// Mitsubishi GX Works2 project: original_finalwithparam   PLC: FX3G

// global labels: Global1
VAR_GLOBAL
  start_day_switch AT X007 : BOOL;
  start_day_light AT Y007 : BOOL;
  cook_switch AT X001 : BOOL;
  cook_is_on_light AT Y001 : BOOL;
  lager_range AT M20 : BOOL;
  pilzner_range AT M19 : BOOL;
  enough_in_pil_stock AT M18 : BOOL;
END_VAR
VAR_GLOBAL CONSTANT
  con_shm_lag : REAL := 150.0;
  con_let_lag : REAL := 12.0;
  con_kash_lag : REAL := 60.0;
  con_shm_pil : REAL := 120.0;
  con_let_pil : REAL := 6.0;
  con_kash_pil : REAL := 53.0;
END_VAR
VAR_GLOBAL
  end_day_light AT M3 : BOOL;
  end_day_switch AT X011 : BOOL;
  shmarim AT D1150 : REAL;
  letet AT D1160 : REAL;
  kashut AT D1170 : REAL;
  analog_input1 AT D8280 : INT;
END_VAR
VAR_GLOBAL CONSTANT
  divide : INT := 400;
  const5 : INT := 5;
END_VAR
VAR_GLOBAL
  input1 AT D1110 : REAL;
  input2 AT D1120 : REAL;
  input3 AT D1130 : REAL;
  Enough_sh_lag AT M50 : BOOL;
  Enough_let_lag AT M51 : BOOL;
  Enough_ksh_lag AT M52 : BOOL;
  const_4 AT K40 : INT;
  Enough_let_pil AT M61 : BOOL;
  Enough_ksh_pil AT M62 : BOOL;
  Enough_sh_pil AT M60 : BOOL;
END_VAR
VAR_GLOBAL CONSTANT
  time_for_fer_const_3S : INT := 30;
  time_for_fer_const_4S : INT := 40;
END_VAR
VAR_GLOBAL
  fert_switch AT X005 : BOOL;
  M_Y3 AT M36 : BOOL;
  Y3_flash_counter AT TC3 : BOOL;
  Y3_light_on AT Y003 : BOOL;
  timer_ts3 AT TS3 : BOOL;
  Y4_flash_counter AT TC4 : BOOL;
  timer_ts4 AT TS4 : BOOL;
  Y4_light_on AT Y004 : BOOL;
  time_fer AT D1140 : INT;
  fert_flash_counter AT TC5 : BOOL;
  fert_flash_counter_ts AT TS5 : BOOL;
  storage_switch AT X002 : BOOL;
  counter_pack AT CC3 : BOOL;
  Y2_light_on AT Y002 : BOOL;
  CC3_term AT CS3 : BOOL;
  reg_pack_count AT D1402 : REAL;
END_VAR
VAR_GLOBAL CONSTANT
  pack_finish : REAL := 1.0;
END_VAR
VAR_GLOBAL
  const_40 AT E40.0 : REAL;
  reg_pack_count_after_multi AT D1404 : REAL;
  analog_output AT D8282 : INT;
  cook_timer AT TC9 : BOOL;
  cook_timer_ts9 AT TS9 : BOOL;
END_VAR
VAR_GLOBAL CONSTANT
  const6 : INT := 6;
END_VAR
VAR_GLOBAL
  help_gate_pil AT M39 : BOOL;
  help_gate_lag AT M38 : BOOL;
  pack_switch AT X000 : BOOL;
  enough_in_lager_stock AT M40 : BOOL;
END_VAR
VAR_GLOBAL CONSTANT
  con_zero : REAL;
END_VAR

// task Task_01 (event TRUE, interval 0, priority 31): POU_01

PROGRAM POU_01
(* structured ladder/FBD written out as ST: instructions are called as NAME(EN, inputs, outputs); _pN, _eN, _tN stand for wires *)
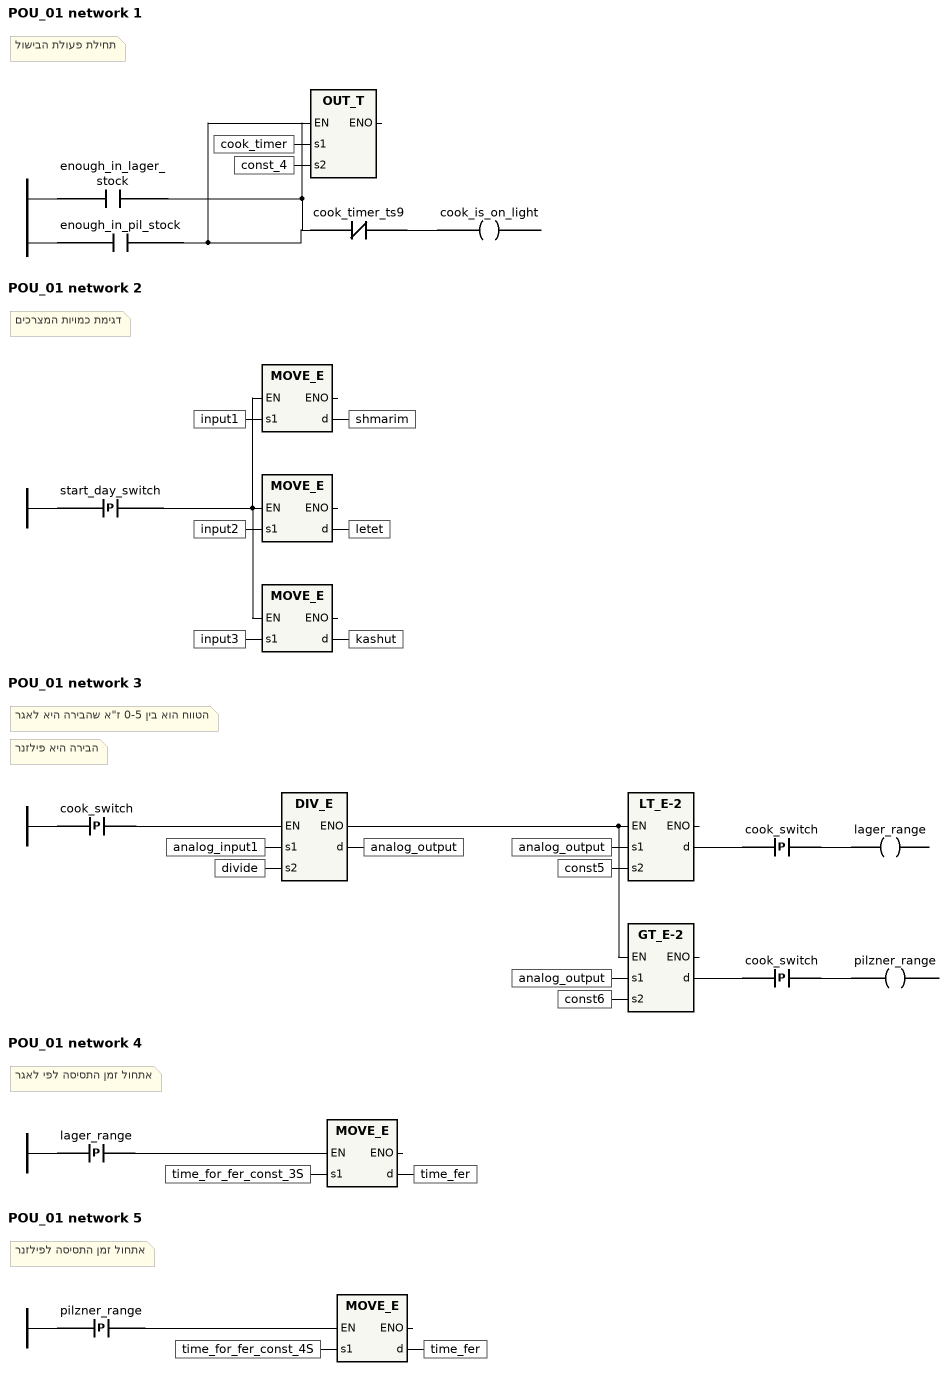
(* network 1 *)
(* תחילת פעולת הבישול *)
_p1 := enough_in_lager_stock OR enough_in_pil_stock;
OUT_T(_p1, cook_timer, const_4);
cook_is_on_light := _p1 AND NOT cook_timer_ts9;
(* network 2 *)
(* דגימת כמויות המצרכים *)
_p1 := LDP(TRUE, start_day_switch);
MOVE_E(_p1, input1, shmarim);
MOVE_E(_p1, input2, letet);
MOVE_E(_p1, input3, kashut);
(* network 3 *)
(* הטווח הוא בין 0-5 ז"א שהבירה היא לאגר *)
(* הבירה היא פילזנר *)
_e1 := DIV_E(LDP(TRUE, cook_switch), analog_input1, divide, analog_output);
LT_E(_e1, analog_output, const5, _t2);
lager_range := _t2 AND LDP(TRUE, cook_switch);
GT_E(_e1, analog_output, const6, _t3);
pilzner_range := _t3 AND LDP(TRUE, cook_switch);
(* network 4 *)
(* אתחול זמן התסיסה לפי לאגר *)
MOVE_E(LDP(TRUE, lager_range), time_for_fer_const_3S, time_fer);
(* network 5 *)
(* אתחול זמן התסיסה לפילזנר *)
MOVE_E(LDP(TRUE, pilzner_range), time_for_fer_const_4S, time_fer);
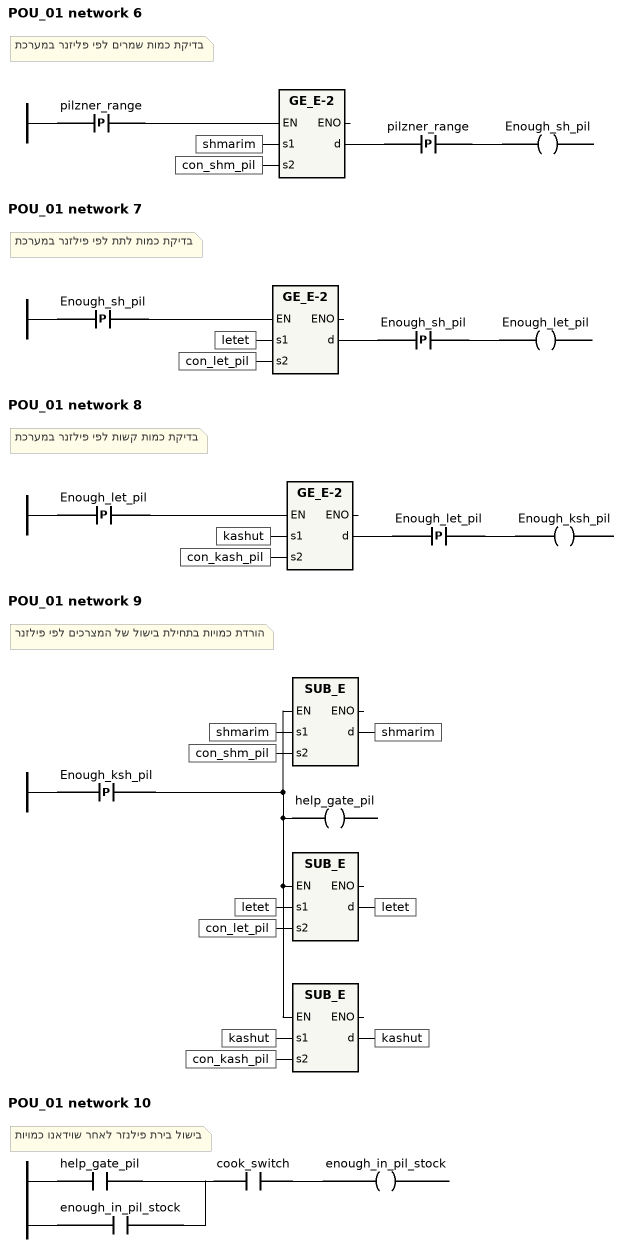
(* network 6 *)
(* בדיקת כמות שמרים לפי פליזנר במערכת *)
GE_E(LDP(TRUE, pilzner_range), shmarim, con_shm_pil, _t1);
Enough_sh_pil := _t1 AND LDP(TRUE, pilzner_range);
(* network 7 *)
(* בדיקת כמות לתת לפי פילזנר במערכת *)
GE_E(LDP(TRUE, Enough_sh_pil), letet, con_let_pil, _t1);
Enough_let_pil := _t1 AND LDP(TRUE, Enough_sh_pil);
(* network 8 *)
(* בדיקת כמות קשות לפי פילזנר במערכת *)
GE_E(LDP(TRUE, Enough_let_pil), kashut, con_kash_pil, _t1);
Enough_ksh_pil := _t1 AND LDP(TRUE, Enough_let_pil);
(* network 9 *)
(* הורדת כמויות בתחילת בישול של המצרכים לפי פילזנר *)
_p1 := LDP(TRUE, Enough_ksh_pil);
help_gate_pil := _p1;
SUB_E(_p1, shmarim, con_shm_pil, shmarim);
SUB_E(_p1, letet, con_let_pil, letet);
SUB_E(_p1, kashut, con_kash_pil, kashut);
(* network 10 *)
(* בישול בירת פילנזר לאחר שוידאנו כמויות *)
enough_in_pil_stock := (help_gate_pil OR enough_in_pil_stock) AND cook_switch;
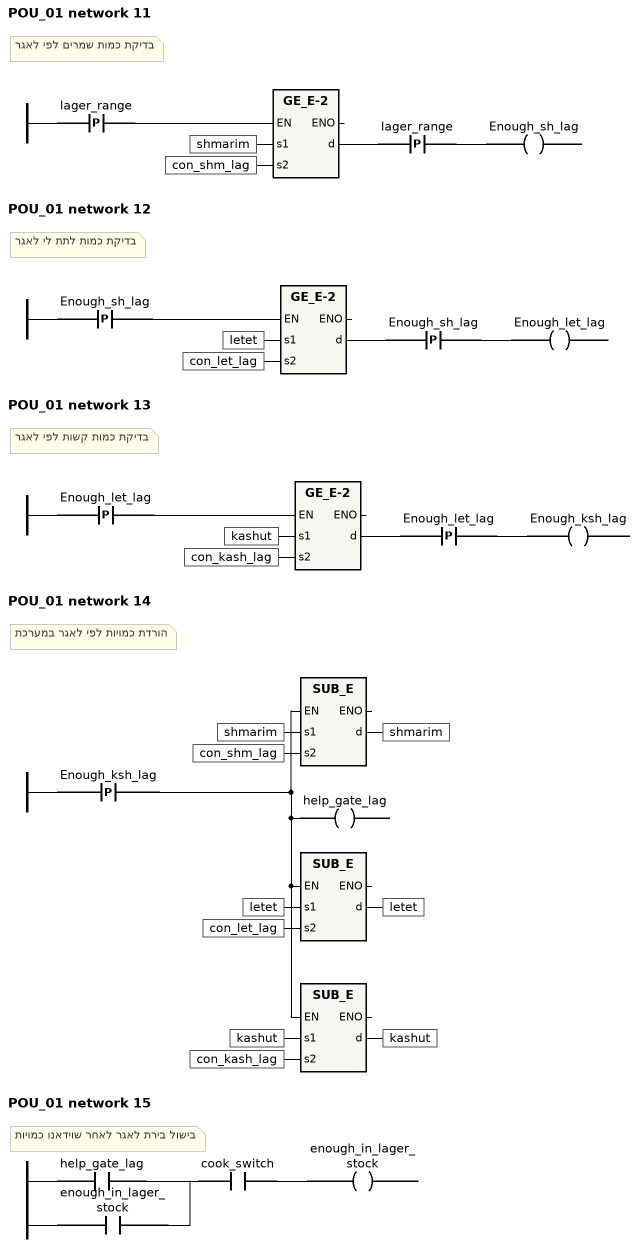
(* network 11 *)
(* בדיקת כמות שמרים לפי לאגר *)
GE_E(LDP(TRUE, lager_range), shmarim, con_shm_lag, _t1);
Enough_sh_lag := _t1 AND LDP(TRUE, lager_range);
(* network 12 *)
(* בדיקת כמות לתת לי לאגר *)
GE_E(LDP(TRUE, Enough_sh_lag), letet, con_let_lag, _t1);
Enough_let_lag := _t1 AND LDP(TRUE, Enough_sh_lag);
(* network 13 *)
(* בדיקת כמות קשות לפי לאגר *)
GE_E(LDP(TRUE, Enough_let_lag), kashut, con_kash_lag, _t1);
Enough_ksh_lag := _t1 AND LDP(TRUE, Enough_let_lag);
(* network 14 *)
(* הורדת כמויות לפי לאגר במערכת *)
_p1 := LDP(TRUE, Enough_ksh_lag);
help_gate_lag := _p1;
SUB_E(_p1, shmarim, con_shm_lag, shmarim);
SUB_E(_p1, letet, con_let_lag, letet);
SUB_E(_p1, kashut, con_kash_lag, kashut);
(* network 15 *)
(* בישול בירת לאגר לאחר שוידאנו כמויות *)
enough_in_lager_stock := (help_gate_lag OR enough_in_lager_stock) AND cook_switch;
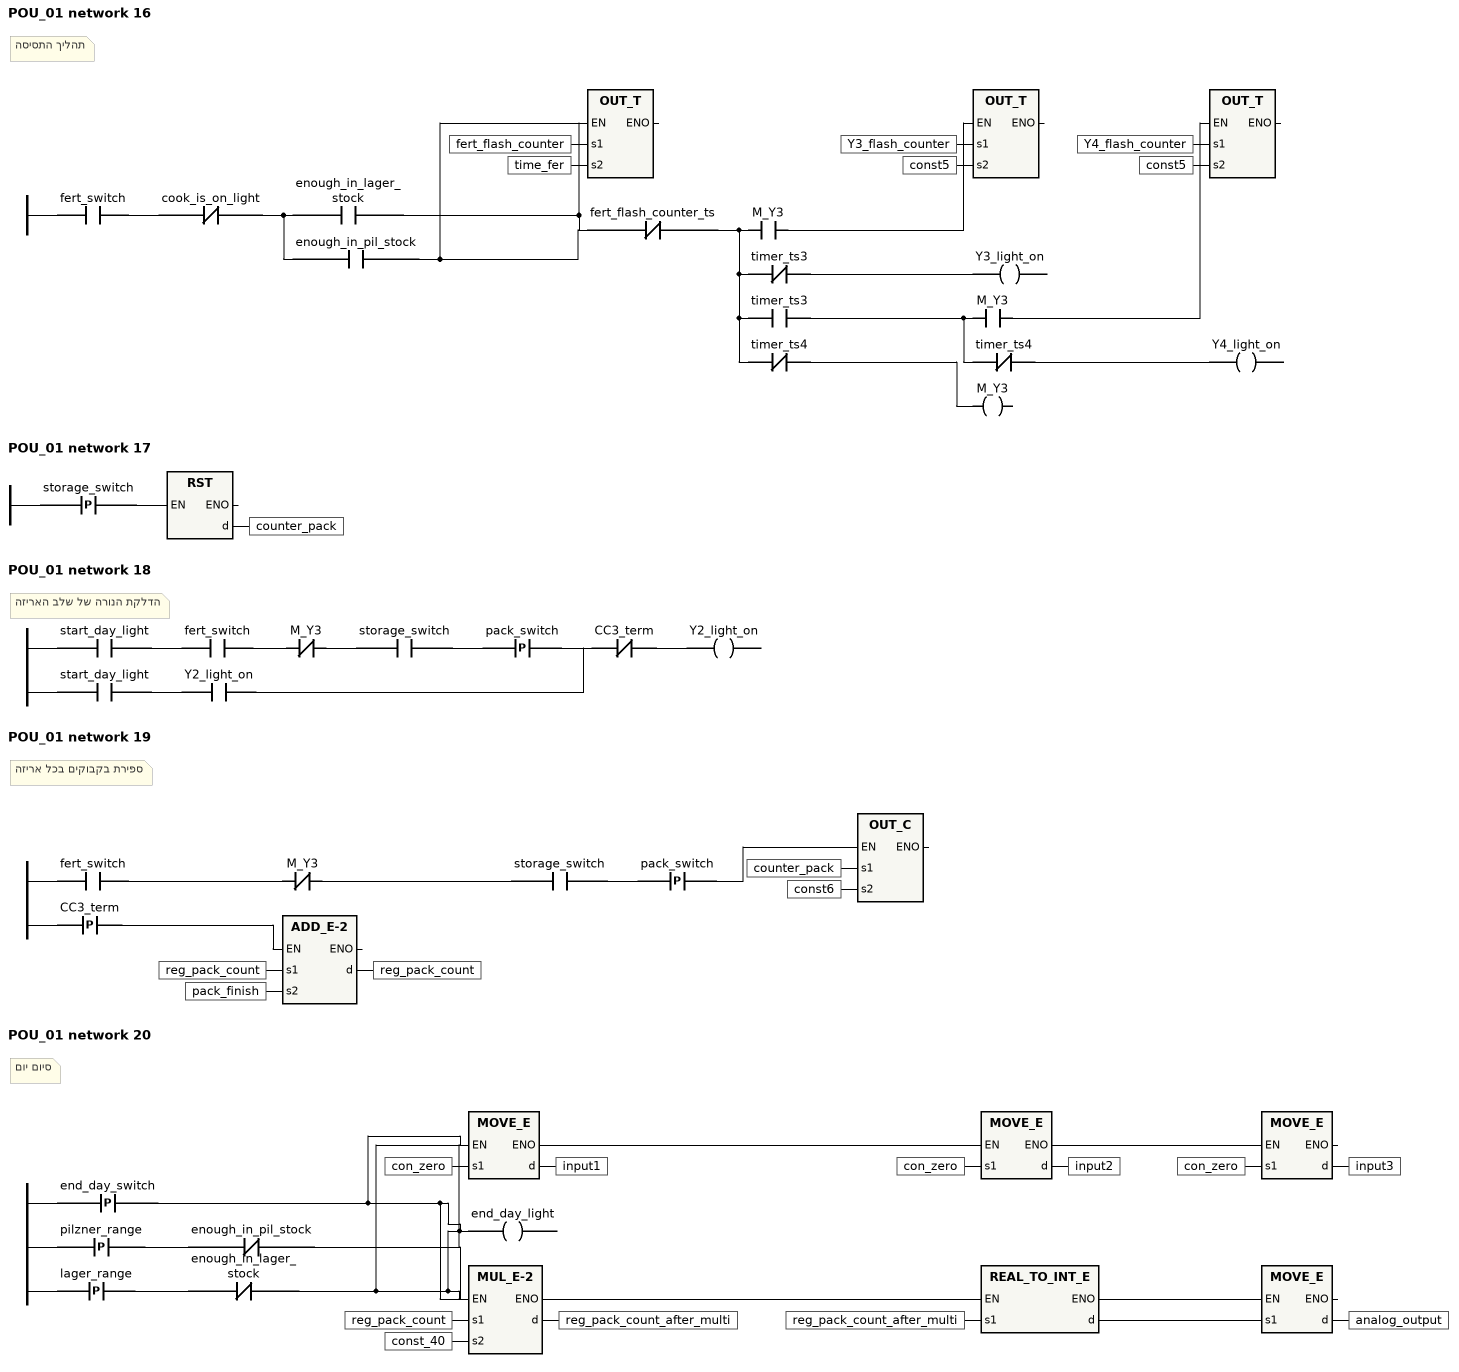
(* network 16 *)
(* תהליך התסיסה *)
_p1 := fert_switch AND NOT cook_is_on_light;
_p2 := (_p1 AND enough_in_lager_stock) OR (_p1 AND enough_in_pil_stock);
OUT_T(_p2, fert_flash_counter, time_fer);
_p3 := _p2 AND NOT fert_flash_counter_ts;
OUT_T(_p3 AND M_Y3, Y3_flash_counter, const5);
Y3_light_on := _p3 AND NOT timer_ts3;
_p4 := _p3 AND timer_ts3;
OUT_T(_p4 AND M_Y3, Y4_flash_counter, const5);
Y4_light_on := _p4 AND NOT timer_ts4;
M_Y3 := _p3 AND NOT timer_ts4;
(* network 17 *)
RST(LDP(TRUE, storage_switch), counter_pack);
(* network 18 *)
(* הדלקת הנורה של שלב האריזה *)
Y2_light_on := ((start_day_light AND fert_switch AND NOT M_Y3 AND storage_switch AND LDP(TRUE, pack_switch)) OR (start_day_light AND Y2_light_on)) AND NOT CC3_term;
(* network 19 *)
(* ספירת בקבוקים בכל אריזה *)
OUT_C(fert_switch AND NOT M_Y3 AND storage_switch AND LDP(TRUE, pack_switch), counter_pack, const6);
ADD_E(LDP(TRUE, CC3_term), reg_pack_count, pack_finish, reg_pack_count);
(* network 20 *)
(* סיום יום *)
_p1 := LDP(TRUE, end_day_switch) OR (LDP(TRUE, pilzner_range) AND NOT enough_in_pil_stock) OR (LDP(TRUE, lager_range) AND NOT enough_in_lager_stock);
end_day_light := _p1;
_e2 := MOVE_E(_p1, con_zero, input1);
_e3 := MOVE_E(_e2, con_zero, input2);
MOVE_E(_e3, con_zero, input3);
_e4 := MUL_E(_p1, reg_pack_count, const_40, reg_pack_count_after_multi);
_e6 := REAL_TO_INT_E(_e4, reg_pack_count_after_multi, _t5);
MOVE_E(_e6, _t5, analog_output);
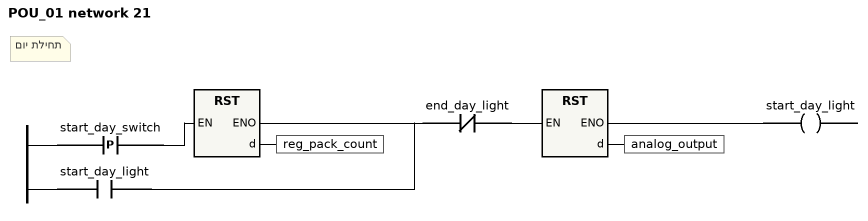
(* network 21 *)
(* תחילת יום *)
_e1 := RST(LDP(TRUE, start_day_switch), reg_pack_count);
_e2 := RST((_e1 OR start_day_light) AND NOT end_day_light, analog_output);
start_day_light := _e2;
END_PROGRAM
